// TIA Portal project "lab-3" (V12)

(* hardware
DEVICE "S7-1200 station_1"  SIMATIC 1200-Station
   slot 0: "S7-1200 rack"  Rack  V1.0
   slot 1: "PLC_1"  CPU 1214C AC/DC/Rly  6ES7 214-1BG31-0XB0  V3.0
      slot 3: "AQ1 x 12 bits_1"  6ES7 232-4HA30-0XB0  V1.0
*)

// ===== PLC "PLC_1"  CPU 1214C AC/DC/Rly =====

VAR_GLOBAL   // PLC tag table "Default tag table"
   "A" AT %M0.0 : Bool;
   "B" AT %M0.1 : Bool;
   "STOP" AT %I0.1 : Bool;
   "START" AT %I0.0 : Bool;
   "START-LATCH" AT %M0.2 : Bool;
   "G" AT %Q0.0 : Bool;
   "Y" AT %Q0.1 : Bool;
   "R" AT %Q0.2 : Bool;
END_VAR

// folder: System blocks/Program resources

DATA_BLOCK "Ty"   // DB1
{ S7_Optimized_Access := 'FALSE' }
AUTHOR : Simatic
FAMILY : IEC
NAME : IEC_TMR
VERSION : 1.0
// stored: InstanceOfName ?
"?"
BEGIN
END_DATA_BLOCK

DATA_BLOCK "Tr"   // DB2
{ S7_Optimized_Access := 'FALSE' }
AUTHOR : Simatic
FAMILY : IEC
NAME : IEC_TMR
VERSION : 1.0
// stored: InstanceOfName ?
"?"
BEGIN
END_DATA_BLOCK

DATA_BLOCK "Tg"   // DB3
{ S7_Optimized_Access := 'FALSE' }
AUTHOR : Simatic
FAMILY : IEC
NAME : IEC_TMR
VERSION : 1.0
// stored: InstanceOfName ?
"?"
BEGIN
END_DATA_BLOCK

// folder: (top level)

ORGANIZATION_BLOCK "Main"   // OB1, LAD, ProgramCycle
TITLE = "Main Program Sweep (Cycle)"
{ S7_Optimized_Access := 'FALSE' }
VERSION : 0.1
   VAR_TEMP   // added for the SCL form of the ladder/FBD networks
      _w1 : Bool;
   END_VAR
BEGIN

REGION Network 1: Start-Stop
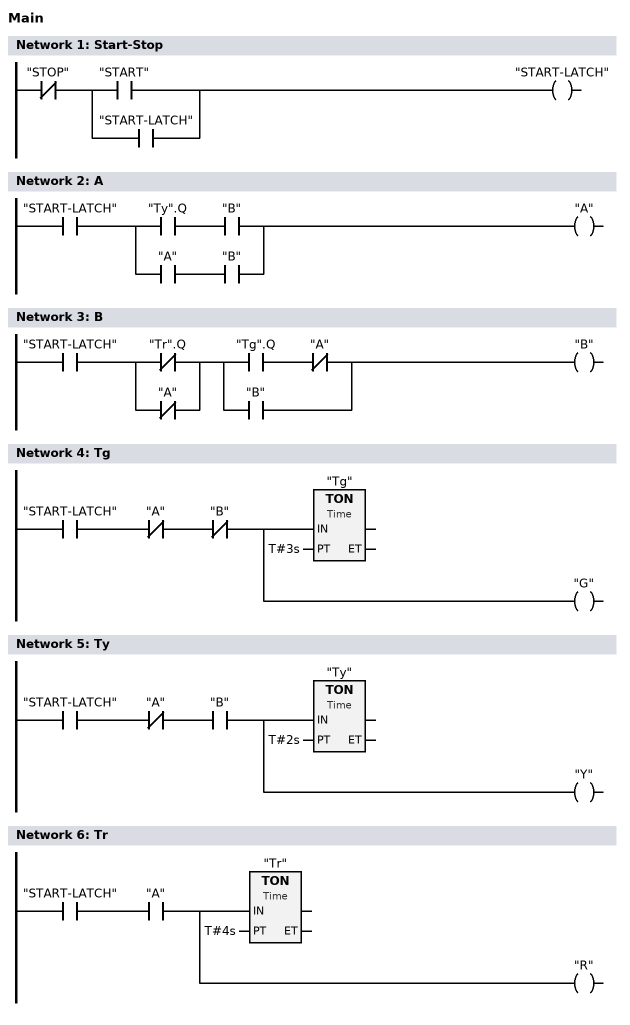
   RUNG wire#powerrail
      I_Contact( "STOP" )
      wire#w1
      Contact( "START" )
      wire#w2
      Coil( "START-LATCH" )
   END_RUNG
   RUNG wire#w1
      Contact( "START-LATCH" )
   END_RUNG wire#w2
   // the same network as SCL:
   "START-LATCH" := NOT "STOP" AND ("START" OR "START-LATCH");
END_REGION

REGION Network 2: A
   RUNG wire#powerrail
      Contact( "START-LATCH" )
      wire#w1
      Contact( "Ty".Q )
      Contact( "B" )
      wire#w2
      Coil( "A" )
   END_RUNG
   RUNG wire#w1
      Contact( "A" )
      Contact( "B" )
   END_RUNG wire#w2
   // the same network as SCL:
   "A" := "START-LATCH" AND (("Ty".Q AND "B") OR ("A" AND "B"));
END_REGION

REGION Network 3: B
   RUNG wire#powerrail
      Contact( "START-LATCH" )
      wire#w1
      I_Contact( "Tr".Q )
      wire#w2
      Contact( "Tg".Q )
      I_Contact( "A" )
      wire#w3
      Coil( "B" )
   END_RUNG
   RUNG wire#w1
      I_Contact( "A" )
   END_RUNG wire#w2
   RUNG wire#w2
      Contact( "B" )
   END_RUNG wire#w3
   // the same network as SCL:
   "B" := "START-LATCH" AND (NOT "Tr".Q OR NOT "A") AND (("Tg".Q AND NOT "A") OR "B");
END_REGION

REGION Network 4: Tg
   #_w1 := "START-LATCH" AND NOT "A" AND NOT "B";
   "Tg".TON(IN := #_w1, PT := T#3s);
   "G" := #_w1;
END_REGION

REGION Network 5: Ty
   #_w1 := "START-LATCH" AND NOT "A" AND "B";
   "Ty".TON(IN := #_w1, PT := T#2s);
   "Y" := #_w1;
END_REGION

REGION Network 6: Tr
   #_w1 := "START-LATCH" AND "A";
   "Tr".TON(IN := #_w1, PT := T#4s);
   "R" := #_w1;
END_REGION
END_ORGANIZATION_BLOCK